Universal Robots PolyScope program: OnRobot_Collision_Detection_Example.urp

Program OnRobot_Collision_Detection_Example (createdIn=3.3.1.237 lastSavedIn=3.7.0.40195 robotSerialNumber=2014359999 directory=/home/ur/ursim-current/programs/TransferVM/Examples/Pendrive installation=default)
Calibrated DH parameters: a=[0.000128, -0.175268, -0.306618, 0.000033, 0.000147, 0]; d=[0.089074, 542.39276, -475.591349, -66.691211, 0.094928, 0.082533]; alpha=[1.570044, -0.000714, -0.003663, 1.570304, -1.570247, 0]; deltaTheta=[0.000007, -1.145705, 0.472188, 0.673551, -0.000038, 0.000057]
BeforeStart
  URCap F/T Zero (FT-OnRobot, OnRobot A/S)
Robot Program (runOnlyOnce=true)
  URCap F/T Guard (FT-OnRobot, OnRobot A/S) dataModel(FX=0.0, FY=0.0, FZ=0.0, TX=0.0, TY=0.0, TZ=0.0, F3D=50.0, T3D=1.0, ABS=true, COORD=0, NAME=50N & 1Nm, OF_PID=4, INDEX=0, STATE=true, ADVANCED=false, NEEDDIGI=false)
    MoveJ speed 60 deg/s, acceleration 80 deg/s^2 (useActiveTCP=false)
      Waypoint Start_WP: TCP in base x=-120.113 y=-431.763 z=146.073 mm, rx=-0.0012 ry=3.1163 rz=0.0389 rad; joints [-91.713, -98.956, -126.223, -46.295, 91.393, -1.776] deg
    URCap F/T Search (FT-OnRobot, OnRobot A/S) dataModel(coordsys=0, absolute=false, advanced=true, speed=0.015, acceleration=0.3, rpy=[0.0, 0.0, 0.0], popupLimit=false, ftarray=[0.0, 0.0, 0.0, 0.0, 0.0, 0.0, 5.0, 0.0], ftabsarray=[false, false, false, false, false, false])
      URCap F/T Waypoint (FT-OnRobot, OnRobot A/S) dataModel(relativeCoords=[0.0, 0.0, -0.05, 0.0, 0.0, 0.0], type=2, z=0.0, x=0.1)
    URCap F/T Move (FT-OnRobot, OnRobot A/S) dataModel(coordsys=0, absolute=false, advanced=true, speed=0.05, acceleration=0.5, rpy=[0.0, 0.0, 0.0], popupLimit=false, ftarray=[0.0, 0.0, 0.0, 0.0, 0.0, 0.0, 5.0, 0.0], ftabsarray=[false, false, false, false, false, false])
      URCap F/T Waypoint (FT-OnRobot, OnRobot A/S) dataModel(relativeCoords=[0.0, 0.0, 0.025, 0.0, 0.0, 0.0], type=2, x=-0.1)
